KUKA KRL program: aip_meta_eki.sub, aip_meta_eki.dat

--- aip_meta_eki.sub ---
&ACCESS RVO1
&REL 48
def aip_meta_eki()
   ; Author: Moritz Weisenboehler (HsKA) <moritz.weisenboehler@hs-karlsruhe.de>

   ;Declarations
   decl int index

   ; Initialization
   ;bas(#initmov, 0)
   init_meta_interface()
   current_meta = null_meta()

   index = 0
   $FLAG[3] = FALSE  ; reset abort_commands flag

   ; Move to current position
   ;ptp $axis_act_meas

   ; Communication process
   loop
      if get_meta(current_meta) then
         ; msgnotify("Recived new meta data", "Meta EKI")
         update_meta(current_meta)
      endif
   endloop
end

deffct meta_type null_meta()
   decl meta_type meta

   meta = { velocity_override 1, abort_commands 0}

   return meta
endfct

def init_meta_interface()
   decl eki_status status
   msgnotify("Init meta interface", "Meta EKI")

   global interrupt decl 17 when $flag[2] == false do close_meta_interface() ;mathias31415 change back to reset_meta_interface()after testing
   interrupt on 17

   global interrupt decl 18 when $timer_flag[2] == true do send_meta_status()
   interrupt on 18

   wait sec 0.012          ; Wait for next interpolation cycle
   $timer[2] = -200        ; Time in [ms] before first interrupt call
   $timer_stop[2] = false  ; Start timer 2

   status = eki_init("AIP_META_EKI")
   status = eki_open("AIP_META_EKI")
end


def reset_meta_interface()
   decl eki_status status
   msgnotify("Reset meta interface", "Meta EKI")

   status = eki_clear("AIP_META_EKI")
   status = eki_init("AIP_META_EKI")
   status = eki_open("AIP_META_EKI")
end

def close_meta_interface()
   decl eki_status status
   msgnotify("Close meta interface", "Meta EKI")
   status = eki_close("AIP_META_EKI")
end


deffct bool has_meta_connection()
   return $flag[2]
endfct


def send_meta_status()
   decl eki_status status

   if has_meta_connection() then
      ;("Send meta status", "Meta EKI")
      ; Command id
      status = eki_setreal("AIP_META_EKI", "MetaState/@VelocityOverride", current_meta.velocity_override)
      status = eki_setint("AIP_META_EKI", "MetaState/@CommandEmpty", 0)

      if has_meta_connection() then
         status = eki_send("AIP_META_EKI", "MetaState")
      endif
   endif

   ; Set timer for next interrupt [ms]
   $timer[2] = -10  ; ~10 ms for above send + 10 ms interrupt timer -> ~50 Hz state transmission
end


def check_error(error_code :in)
   decl int error_code

   decl char error_message[64]
   decl int index

   index = 0

   for index = 1 to 64
      error_message[index] = " "
   endfor

   if error_code > 0 then
      switch error_code
         case 1
            error_message[] = "Fehler 1"
         default
            error_message[] = "Unbekannter Fehler"
      endswitch

      send_error(error_code, error_message[])
     endif
end

def send_error(error_code :in, error_message[] :in)
   decl int error_code
   decl char error_message[]

   decl eki_status status

   if has_meta_connection() then
      status = eki_setint("AIP_META_EKI", "MetaState/Error/@Code", error_code)
      status = eki_setstring("AIP_META_EKI", "MetaState/Error/@Message", error_message[])
   endif
end


deffct bool has_meta()
   decl eki_status status

   if not has_meta_connection() then
      return false
   endif

   status = eki_checkbuffer("AIP_META_EKI", "MetaCommand/@VelocityOverride")

   return status.buff > 0
endfct


deffct bool get_meta(meta :out)
   decl meta_type meta

   decl eki_status status

   if not has_meta() then
     return false
   endif

   status = eki_getreal("AIP_META_EKI", "MetaCommand/@VelocityOverride", meta.velocity_override)
   status = eki_getint("AIP_META_EKI", "MetaCommand/@AbortCommands", meta.abort_commands)

   return true
endfct


def update_meta(meta :in)
   decl meta_type meta
   ; Update velocity_override
   ; msgnotify("Handeling for velocity_override not implemented. Recived velocity_override: %1 ",,meta.velocity_override)

   ; Update abort_commands_flag
   if meta.abort_commands == 1 then
      $FLAG[3] = TRUE
      msgnotify("Set abort_commands flag ($FLAG[3]) to TRUE", "Meta EKI")
   else
      $FLAG[3] = FALSE
      msgnotify("Set abort_commands flag ($FLAG[3]) to FALSE", "Meta EKI")
   endif
end

--- aip_meta_eki.dat ---
&ACCESS RVO
&REL 48
defdat aip_meta_eki
   struc meta_type real velocity_override, int abort_commands
   decl meta_type current_meta
enddat
